SUBAPPLICATION Uebung_035a (* Ampelschaltung International *)
  (* Standard: 61499-2; Description: Copyright (c) 2023 Meisterschulen am Ostbahnhof This program and the accompanying materials are made available under the terms of the Eclipse Public License 2.0 which is available at https://www.eclipse.org/legal/epl-2.0/ SPDX-License-Identifier: EPL-2.0 *)
  (* Version 1.0, 2023-10-23, Franz Höpfinger, Meisterschulen am Ostbahnhof *)
  PACKAGE Uebungen;
  IMPORT logiBUS::io::DI::logiBUS_DI::Input_I1;
  IMPORT logiBUS::io::DI::logiBUS_DI_Events::BUTTON_SINGLE_CLICK;
  IMPORT logiBUS::io::DQ::logiBUS_DO::Output_Q1;
  IMPORT logiBUS::io::DQ::logiBUS_DO::Output_Q2;
  IMPORT logiBUS::io::DQ::logiBUS_DO::Output_Q3;
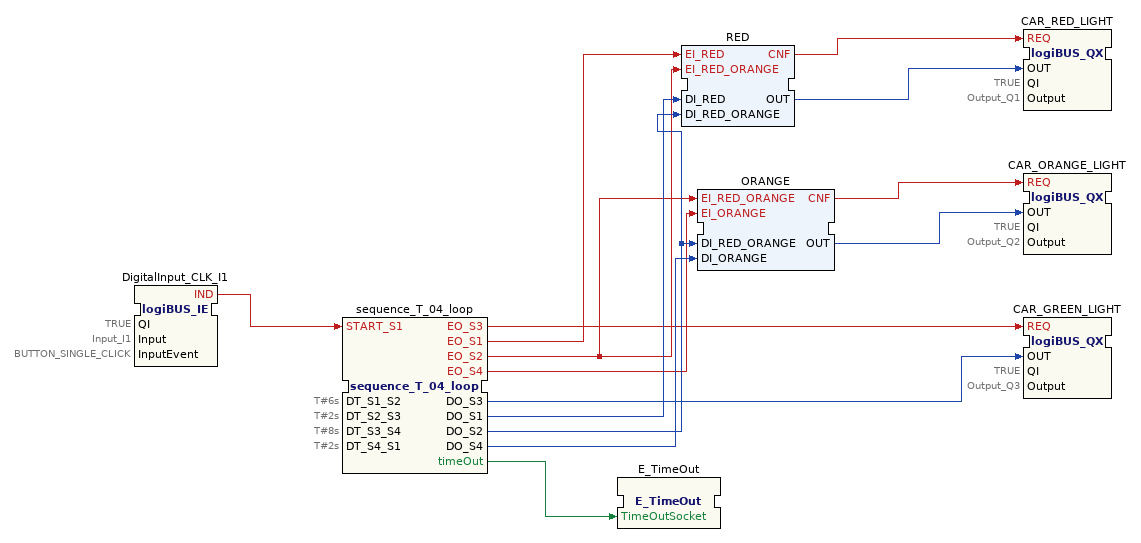
  FBS
    CAR_RED_LIGHT : logiBUS::io::DQ::logiBUS_QX(QI := TRUE, Output := Output_Q1);
    E_TimeOut : iec61499::events::E_TimeOut;
    CAR_ORANGE_LIGHT : logiBUS::io::DQ::logiBUS_QX(QI := TRUE, Output := Output_Q2);
    CAR_GREEN_LIGHT : logiBUS::io::DQ::logiBUS_QX(QI := TRUE, Output := Output_Q3);
    DigitalInput_CLK_I1 : logiBUS::io::DI::logiBUS_IE(QI := TRUE, Input := Input_I1, InputEvent := BUTTON_SINGLE_CLICK);
    sequence_T_04_loop : logiBUS::utils::sequence::timed::sequence_T_04_loop(DT_S1_S2 := T#6s (* RED *), DT_S2_S3 := T#2s (* RED+ORANGE *), DT_S3_S4 := T#8s (* GREEN *), DT_S4_S1 := T#2s (* ORANGE *), EO_S1 :=  (* RED *), EO_S2 :=  (* RED+ORANGE *), EO_S3 :=  (* GREEN *), EO_S4 :=  (* ORANGE *), DO_S1 :=  (* RED *), DO_S2 :=  (* RED+ORANGE *), DO_S3 :=  (* GREEN *), DO_S4 :=  (* ORANGE *));
  END_FBS
  SUBAPPLICATION RED
    EVENT_INPUT
      EI_RED;
      EI_RED_ORANGE;
    END_EVENT
    EVENT_OUTPUT
      CNF;
    END_EVENT
    VAR_INPUT
      DI_RED : ANY_BIT;
      DI_RED_ORANGE : ANY_BIT;
    END_VAR
    VAR_OUTPUT
      OUT : ANY_BIT;
    END_VAR
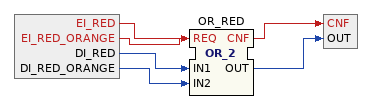
    FBS
      OR_RED : iec61131::bitwiseOperators::OR_2;
    END_FBS
    EVENT_CONNECTIONS
      EI_RED TO OR_RED.REQ;
      EI_RED_ORANGE TO OR_RED.REQ;
      OR_RED.CNF TO CNF;
    END_CONNECTIONS
    DATA_CONNECTIONS
      DI_RED TO OR_RED.IN1;
      DI_RED_ORANGE TO OR_RED.IN2;
      OR_RED.OUT TO OUT;
    END_CONNECTIONS
  END_SUBAPPLICATION
  SUBAPPLICATION ORANGE
    EVENT_INPUT
      EI_RED_ORANGE;
      EI_ORANGE;
    END_EVENT
    EVENT_OUTPUT
      CNF;
    END_EVENT
    VAR_INPUT
      DI_RED_ORANGE : ANY_BIT;
      DI_ORANGE : ANY_BIT;
    END_VAR
    VAR_OUTPUT
      OUT : ANY_BIT;
    END_VAR
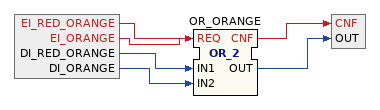
    FBS
      OR_ORANGE : iec61131::bitwiseOperators::OR_2;
    END_FBS
    EVENT_CONNECTIONS
      EI_RED_ORANGE TO OR_ORANGE.REQ;
      EI_ORANGE TO OR_ORANGE.REQ;
      OR_ORANGE.CNF TO CNF;
    END_CONNECTIONS
    DATA_CONNECTIONS
      DI_RED_ORANGE TO OR_ORANGE.IN1;
      DI_ORANGE TO OR_ORANGE.IN2;
      OR_ORANGE.OUT TO OUT;
    END_CONNECTIONS
  END_SUBAPPLICATION
  EVENT_CONNECTIONS
    DigitalInput_CLK_I1.IND TO sequence_T_04_loop.START_S1;
    sequence_T_04_loop.EO_S3 TO CAR_GREEN_LIGHT.REQ;
    sequence_T_04_loop.EO_S1 TO RED.EI_RED;
    sequence_T_04_loop.EO_S2 TO RED.EI_RED_ORANGE;
    RED.CNF TO CAR_RED_LIGHT.REQ;
    sequence_T_04_loop.EO_S2 TO ORANGE.EI_RED_ORANGE;
    sequence_T_04_loop.EO_S4 TO ORANGE.EI_ORANGE;
    ORANGE.CNF TO CAR_ORANGE_LIGHT.REQ;
  END_CONNECTIONS
  DATA_CONNECTIONS
    sequence_T_04_loop.DO_S3 TO CAR_GREEN_LIGHT.OUT;
    sequence_T_04_loop.DO_S1 TO RED.DI_RED;
    sequence_T_04_loop.DO_S2 TO RED.DI_RED_ORANGE;
    RED.OUT TO CAR_RED_LIGHT.OUT;
    sequence_T_04_loop.DO_S2 TO ORANGE.DI_RED_ORANGE;
    sequence_T_04_loop.DO_S4 TO ORANGE.DI_ORANGE;
    ORANGE.OUT TO CAR_ORANGE_LIGHT.OUT;
  END_CONNECTIONS
  ADAPTER_CONNECTIONS
    sequence_T_04_loop.timeOut TO E_TimeOut.TimeOutSocket;
  END_CONNECTIONS
END_SUBAPPLICATION
